(* PLC project cmd_motor_2d1s, Dassault Systèmes ControlBuild 2024x *)
(* stored: creationDateTime 2023-10-03T11:13:34-01:00 *)

FUNCTION_BLOCK actuator
  VAR_INPUT
    autoMode : BOOL := false;
    manualMode : BOOL := false;
  END_VAR
  VAR_INPUT
    autoFwdCmd : BOOL := false;
    autoBwdCmd : BOOL := false;
  END_VAR
  VAR_INPUT
    forwardPB : BOOL := false;
    backwardPB : BOOL := false;
    offPB : BOOL := false;
  END_VAR
  VAR_INPUT
    generalFault : BOOL := false;
  END_VAR
  VAR_OUTPUT
    backwardCmd : BOOL := false;
    forwardCmd : BOOL := false;
  END_VAR

(* LD diagram, written out as Structured Text *)
1:
forwardCmd := (autoMode AND autoFwdCmd OR manualMode AND (forwardCmd OR forwardPB AND NOT backwardPB) AND NOT offPB AND NOT backwardCmd) AND NOT generalFault;
2:
backwardCmd := (autoMode AND autoBwdCmd OR manualMode AND (backwardCmd OR backwardPB AND NOT forwardPB) AND NOT offPB AND NOT forwardCmd) AND NOT generalFault;
END_FUNCTION_BLOCK

FUNCTION_BLOCK faults
  VAR_INPUT
    forwardCmd : BOOL := false;
    backwardCmd : BOOL := false;
  END_VAR
  VAR_INPUT
    thermalFB : BOOL := false;
    forwardFB : BOOL := false;
    backwardFB : BOOL := false;
  END_VAR
  VAR_INPUT
    acknowledgePB : BOOL := false;
  END_VAR
  VAR_OUTPUT
    generalFault : BOOL := false;
  END_VAR
  VAR
    thermalFault : BOOL := false;
    forwardFBFault : BOOL := false;
    backwardFBFault : BOOL := false;
  END_VAR

(* LD diagram, written out as Structured Text *)
1:
IF acknowledgePB THEN thermalFault := FALSE; END_IF;
IF acknowledgePB THEN forwardFBFault := FALSE; END_IF;
IF acknowledgePB THEN backwardFBFault := FALSE; END_IF;
IF acknowledgePB THEN generalFault := FALSE; END_IF;
2:
TON_FW(IN := forwardCmd, PT := T#0h0m2s0ms);
IF TON_FW.Q0 AND NOT forwardFB THEN forwardFBFault := TRUE; END_IF;
TON_BW(IN := backwardCmd, PT := T#0h0m2s0ms);
IF TON_BW.Q0 AND NOT backwardFB THEN backwardFBFault := TRUE; END_IF;
3:
IF NOT thermalFB THEN thermalFault := TRUE; END_IF;
4:
IF thermalFault OR forwardFBFault OR backwardFBFault THEN generalFault := TRUE; END_IF;
END_FUNCTION_BLOCK

(* Command of a motor with two directions and one speed and with fault detection *)
PROGRAM cmd_equipment_library.cmd_motor_2d1s
  VAR_INPUT
    autoMode : BOOL := false;
    manualMode : BOOL := false;
  END_VAR
  VAR_INPUT
    autoFwdCmd : BOOL := false;
    autoBwdCmd : BOOL := false;
  END_VAR
  VAR_INPUT
    forwardPB : BOOL := false;
    backwardPB : BOOL := false;
    stopPB : BOOL := false;
  END_VAR
  VAR_INPUT
    thermalFB : BOOL := false;
    forwardFB : BOOL := false;
    backwardFB : BOOL := false;
  END_VAR
  VAR_INPUT
    acknowledgePB : BOOL := false;
  END_VAR
  VAR_OUTPUT
    forwardCmd : BOOL := false;
    backwardCmd : BOOL := false;
  END_VAR
  VAR_OUTPUT
    generalFault : BOOL := false;
  END_VAR

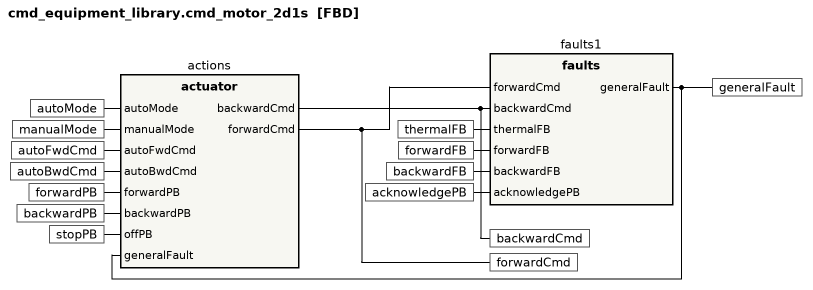
(* FBD diagram, written out as Structured Text *)
faults1(forwardCmd := actions.forwardCmd, backwardCmd := actions.backwardCmd, thermalFB := thermalFB, forwardFB := forwardFB, backwardFB := backwardFB, acknowledgePB := acknowledgePB);
actions(autoMode := autoMode, manualMode := manualMode, autoFwdCmd := autoFwdCmd, autoBwdCmd := autoBwdCmd, forwardPB := forwardPB, backwardPB := backwardPB, offPB := stopPB, generalFault := faults1.generalFault);
forwardCmd := actions.forwardCmd;
backwardCmd := actions.backwardCmd;
generalFault := faults1.generalFault;
END_PROGRAM
